LIN {X 0,Y 55.699,Z 480.431,A -85,B 0,C 180,E1 -29739.752,E2 -29739.752} C_VEL
LIN {X 0,Y 58.966,Z 465.331,A -85,B 0,C 180,E1 -29745.097,E2 -29745.097} C_VEL
LIN {X 0,Y 62.169,Z 448.108,A -85,B 0,C 180,E1 -29749.414,E2 -29749.414} C_VEL
LIN {X 0,Y 73.218,Z 385.483,A -85,B 0,C 180,E1 -29760.921,E2 -29760.921} C_VEL
LIN {X 0,Y 72.492,Z 382.499,A -85,B 0,C 180,E1 -29761.896,E2 -29761.896} C_VEL
LIN {X 0,Y 69.464,Z 373.63,A -85,B 0,C 180,E1 -29765.325,E2 -29765.325} C_VEL
LIN {X 0,Y 67.284,Z 368.876,A -85,B 0,C 180,E1 -29767.632,E2 -29767.632} C_VEL
LIN {X 0,Y 64.336,Z 364.78,A -85,B 0,C 180,E1 -29770.407,E2 -29770.407} C_VEL
LIN {X 0,Y 57.379,Z 355.76,A -85,B 0,C 180,E1 -29778.129,E2 -29778.129} C_VEL
LIN {X 0,Y 55.471,Z 351.155,A -85,B 0,C 180,E1 -29781.461,E2 -29781.461} C_VEL
LIN {X 0,Y 51.666,Z 340.966,A -85,B 0,C 180,E1 -29789.989,E2 -29789.989} C_VEL
LIN {X 0,Y 48.729,Z 333.984,A -85,B 0,C 180,E1 -29798.281,E2 -29798.281} C_VEL
LIN {X 0,Y 46.247,Z 330.846,A -85,B 0,C 180,E1 -29805.867,E2 -29805.867} C_VEL
LIN {X 0,Y 45.665,Z 329.617,A -85,B 0,C 180,E1 -29808.495,E2 -29808.495} C_VEL
LIN {X 0,Y 42.859,Z 326.9,A -85,B 0,C 180,E1 -29824.939,E2 -29824.939} C_VEL
LIN {X 0,Y 42.565,Z 326.431,A -85,B 0,C 180,E1 -29831.316,E2 -29831.316} C_VEL
LIN {X 0,Y 42.67,Z 326.804,A -85,B 0,C 180,E1 -29840.533,E2 -29840.533} C_VEL
LIN {X 0,Y 43.226,Z 327.728,A -85,B 0,C 180,E1 -29847.197,E2 -29847.197} C_VEL
LIN {X 0,Y 45.942,Z 330.085,A -85,B 0,C 180,E1 -29860.528,E2 -29860.528} C_VEL
LIN {X 0,Y 47.787,Z 333.251,A -85,B 0,C 180,E1 -29867.187,E2 -29867.187} C_VEL
LIN {X 0,Y 49.086,Z 334.684,A -85,B 0,C 180,E1 -29870.587,E2 -29870.587} C_VEL
LIN {X 0,Y 51.573,Z 340.348,A -85,B 0,C 180,E1 -29877.378,E2 -29877.378} C_VEL
LIN {X 0,Y 55.316,Z 350.367,A -85,B 0,C 180,E1 -29885.909,E2 -29885.909} C_VEL
LIN {X 0,Y 59.591,Z 363.131,A -85,B 0,C 180,E1 -29893.866,E2 -29893.866} C_VEL
LIN {X 0,Y 63.329,Z 378.635,A -85,B 0,C 180,E1 -29900.74,E2 -29900.74} C_VEL
LIN {X 0,Y 67.376,Z 395.193,A -85,B 0,C 180,E1 -29906.947,E2 -29906.947} C_VEL
LIN {X 0,Y 54.893,Z 463.552,A -85,B 0,C 180,E1 -29921.285,E2 -29921.285} C_VEL
LIN {X 0,Y 51.895,Z 478.587,A -85,B 0,C 180,E1 -29926.34,E2 -29926.34} C_VEL
LIN {X 0,Y 48.679,Z 493.737,A -85,B 0,C 180,E1 -29933.463,E2 -29933.463} C_VEL
LIN {X 0,Y 45.63,Z 509.372,A -85,B 0,C 180,E1 -29943.73,E2 -29943.73} C_VEL
LIN {X 0,Y 44.068,Z 522.69,A -85,B 0,C 180,E1 -29955.453,E2 -29955.453} C_VEL
LIN {X 0,Y 44.336,Z 534.77,A -85,B 0,C 180,E1 -29968.467,E2 -29968.467} C_VEL
LIN {X 0,Y 46.533,Z 544.973,A -85,B 0,C 180,E1 -29980.894,E2 -29980.894} C_VEL
LIN {X 0,Y 48.842,Z 550.837,A -85,B 0,C 180,E1 -29988.592,E2 -29988.592} C_VEL
LIN {X 0,Y 49.64,Z 553.845,A -85,B 0,C 180,E1 -29995.146,E2 -29995.146} C_VEL
LIN {X 0,Y 53.747,Z 560.113,A -85,B 0,C 180,E1 -30010.842,E2 -30010.842} C_VEL
LIN {X 0,Y 54.729,Z 560.872,A -85,B 0,C 180,E1 -30015.059,E2 -30015.059} C_VEL
LIN {X 0,Y 46.975,Z 550.464,A -85,B 0,C 180,E1 -30030.899,E2 -30030.899} C_VEL
LIN {X 0,Y 44.588,Z 544.97,A -85,B 0,C 180,E1 -30039.221,E2 -30039.221} C_VEL
LIN {X 0,Y 42.294,Z 536.859,A -85,B 0,C 180,E1 -30050.427,E2 -30050.427} C_VEL
LIN {X 0,Y 41.213,Z 525.272,A -85,B 0,C 180,E1 -30064.884,E2 -30064.884} C_VEL
LIN {X 0,Y 42.221,Z 511.198,A -85,B 0,C 180,E1 -30079.438,E2 -30079.438} C_VEL
LIN {X 0,Y 45.13,Z 495.507,A -85,B 0,C 180,E1 -30091.699,E2 -30091.699} C_VEL
LIN {X 0,Y 48.94,Z 478.571,A -85,B 0,C 180,E1 -30101.013,E2 -30101.013} C_VEL
LIN {X 0,Y 52.42,Z 462.754,A -85,B 0,C 180,E1 -30107.03,E2 -30107.03} C_VEL
LIN {X 0,Y 56.128,Z 443.14,A -85,B 0,C 180,E1 -30112.214,E2 -30112.214} C_VEL
LIN {X 0,Y 66.667,Z 386.304,A -85,B 0,C 180,E1 -30123.427,E2 -30123.427} C_VEL
LIN {X 0,Y 60.039,Z 364.937,A -85,B 0,C 180,E1 -30133.113,E2 -30133.113} C_VEL
LIN {X 0,Y 56.099,Z 352.921,A -85,B 0,C 180,E1 -30140.227,E2 -30140.227} C_VEL
LIN {X 0,Y 55.471,Z 351.155,A -85,B 0,C 180,E1 -30141.461,E2 -30141.461} C_VEL
LIN {X 0,Y 54.149,Z 348.336,A -85,B 0,C 180,E1 -30143.904,E2 -30143.904} C_VEL
LIN {X 0,Y 52.232,Z 346.304,A -85,B 0,C 180,E1 -30146.934,E2 -30146.934} C_VEL
LIN {X 0,Y 46.327,Z 341.623,A -85,B 0,C 180,E1 -30158.375,E2 -30158.375} C_VEL
LIN {X 0,Y 45.874,Z 340.912,A -85,B 0,C 180,E1 -30159.735,E2 -30159.735} C_VEL
LIN {X 0,Y 45.049,Z 339.451,A -85,B 0,C 180,E1 -30162.557,E2 -30162.557} C_VEL
LIN {X 0,Y 43.071,Z 336.15,A -85,B 0,C 180,E1 -30170.881,E2 -30170.881} C_VEL
LIN {X 0,Y 40.853,Z 333.573,A -85,B 0,C 180,E1 -30187.874,E2 -30187.874} C_VEL
LIN {X 0,Y 40.719,Z 333.35,A -85,B 0,C 180,E1 -30193.642,E2 -30193.642} C_VEL
LIN {X 0,Y 41.056,Z 333.988,A -85,B 0,C 180,E1 -30203.361,E2 -30203.361} C_VEL
LIN {X 0,Y 43.333,Z 336.653,A -85,B 0,C 180,E1 -30218.203,E2 -30218.203} C_VEL
LIN {X 0,Y 45.356,Z 339.979,A -85,B 0,C 180,E1 -30226.322,E2 -30226.322} C_VEL
LIN {X 0,Y 46.092,Z 341.294,A -85,B 0,C 180,E1 -30228.723,E2 -30228.723} C_VEL
LIN {X 0,Y 48.368,Z 347.727,A -85,B 0,C 180,E1 -30236.318,E2 -30236.318} C_VEL
LIN {X 0,Y 51.301,Z 357.024,A -85,B 0,C 180,E1 -30244.306,E2 -30244.306} C_VEL
LIN {X 0,Y 54.68,Z 368.265,A -85,B 0,C 180,E1 -30251.748,E2 -30251.748} C_VEL
LIN {X 0,Y 59.813,Z 392.087,A -85,B 0,C 180,E1 -30262.664,E2 -30262.664} C_VEL
LIN {X 0,Y 60.736,Z 395.951,A -85,B 0,C 180,E1 -30264.231,E2 -30264.231} C_VEL
LIN {X 0,Y 48.122,Z 462.205,A -85,B 0,C 180,E1 -30279.548,E2 -30279.548} C_VEL
LIN {X 0,Y 44.955,Z 477.483,A -85,B 0,C 180,E1 -30285.309,E2 -30285.309} C_VEL
LIN {X 0,Y 41.591,Z 492.983,A -85,B 0,C 180,E1 -30293.759,E2 -30293.759} C_VEL
LIN {X 0,Y 38.707,Z 508.521,A -85,B 0,C 180,E1 -30305.932,E2 -30305.932} C_VEL
LIN {X 0,Y 37.602,Z 521.263,A -85,B 0,C 180,E1 -30319.243,E2 -30319.243} C_VEL
LIN {X 0,Y 38.441,Z 532.103,A -85,B 0,C 180,E1 -30332.634,E2 -30332.634} C_VEL
LIN {X 0,Y 41.041,Z 541.3,A -85,B 0,C 180,E1 -30344.898,E2 -30344.898} C_VEL
LIN {X 0,Y 43.949,Z 547.593,A -85,B 0,C 180,E1 -30353.578,E2 -30353.578} C_VEL
LIN {X 0,Y 45.292,Z 550.922,A -85,B 0,C 180,E1 -30361.936,E2 -30361.936} C_VEL
LIN {X 0,Y 46.545,Z 552.86,A -85,B 0,C 180,E1 -30367.17,E2 -30367.17} C_VEL
LIN {X 0,Y 48.338,Z 554.843,A -85,B 0,C 180,E1 -30373.359,E2 -30373.359} C_VEL
LIN {X 0,Y 41.402,Z 545.488,A -85,B 0,C 180,E1 -30388.1,E2 -30388.1} C_VEL
LIN {X 0,Y 38.272,Z 538.77,A -85,B 0,C 180,E1 -30398.444,E2 -30398.444} C_VEL
LIN {X 0,Y 35.716,Z 529.842,A -85,B 0,C 180,E1 -30411.507,E2 -30411.507} C_VEL
LIN {X 0,Y 34.889,Z 518.192,A -85,B 0,C 180,E1 -30427.223,E2 -30427.223} C_VEL
LIN {X 0,Y 36.013,Z 505.529,A -85,B 0,C 180,E1 -30441.454,E2 -30441.454} C_VEL
LIN {X 0,Y 38.612,Z 492.029,A -85,B 0,C 180,E1 -30453.086,E2 -30453.086} C_VEL
LIN {X 0,Y 42.449,Z 475.565,A -85,B 0,C 180,E1 -30463.064,E2 -30463.064} C_VEL
LIN {X 0,Y 46.079,Z 459.423,A -85,B 0,C 180,E1 -30469.683,E2 -30469.683} C_VEL
LIN {X 0,Y 51.287,Z 432.312,A -85,B 0,C 180,E1 -30477.057,E2 -30477.057} C_VEL
LIN {X 0,Y 60.147,Z 387.558,A -85,B 0,C 180,E1 -30486.307,E2 -30486.307} C_VEL
LIN {X 0,Y 54.234,Z 367.063,A -85,B 0,C 180,E1 -30496.882,E2 -30496.882} C_VEL
LIN {X 0,Y 50.513,Z 354.677,A -85,B 0,C 180,E1 -30505.432,E2 -30505.432} C_VEL
LIN {X 0,Y 47.276,Z 344.825,A -85,B 0,C 180,E1 -30514.818,E2 -30514.818} C_VEL
LIN {X 0,Y 45.874,Z 340.912,A -85,B 0,C 180,E1 -30519.735,E2 -30519.735} C_VEL
LIN {X 0,Y 44.694,Z 339.743,A -85,B 0,C 180,E1 -30523.229,E2 -30523.229} C_VEL
LIN {X 0,Y 42.755,Z 339.599,A -85,B 0,C 180,E1 -30528.729,E2 -30528.729} C_VEL
LIN {X 0,Y 39.587,Z 340.945,A -85,B 0,C 180,E1 -30541.368,E2 -30541.368} C_VEL
LIN {X 0,Y 39.05,Z 340.575,A -85,B 0,C 180,E1 -30547.31,E2 -30547.31} C_VEL
LIN {X 0,Y 38.927,Z 340.263,A -85,B 0,C 180,E1 -30556.212,E2 -30556.212} C_VEL
LIN {X 0,Y 39.266,Z 341.215,A -85,B 0,C 180,E1 -30564.444,E2 -30564.444} C_VEL
LIN {X 0,Y 40.791,Z 343.118,A -85,B 0,C 180,E1 -30575.645,E2 -30575.645} C_VEL
LIN {X 0,Y 42.632,Z 346.581,A -85,B 0,C 180,E1 -30584.499,E2 -30584.499} C_VEL
LIN {X 0,Y 44.258,Z 352.215,A -85,B 0,C 180,E1 -30591.784,E2 -30591.784} C_VEL
LIN {X 0,Y 46.576,Z 361.026,A -85,B 0,C 180,E1 -30600.249,E2 -30600.249} C_VEL
LIN {X 0,Y 49.278,Z 371.489,A -85,B 0,C 180,E1 -30608.031,E2 -30608.031} C_VEL
LIN {X 0,Y 54.241,Z 396.884,A -85,B 0,C 180,E1 -30621.036,E2 -30621.036} C_VEL
LIN {X 0,Y 41.251,Z 461.358,A -85,B 0,C 180,E1 -30637.528,E2 -30637.528} C_VEL
LIN {X 0,Y 37.971,Z 476.59,A -85,B 0,C 180,E1 -30644.196,E2 -30644.196} C_VEL
LIN {X 0,Y 34.373,Z 492.897,A -85,B 0,C 180,E1 -30654.885,E2 -30654.885} C_VEL
LIN {X 0,Y 31.868,Z 507.771,A -85,B 0,C 180,E1 -30669.389,E2 -30669.389} C_VEL
LIN {X 0,Y 31.573,Z 521.341,A -85,B 0,C 180,E1 -30686.827,E2 -30686.827} C_VEL
LIN {X 0,Y 34.309,Z 533.798,A -85,B 0,C 180,E1 -30704.852,E2 -30704.852} C_VEL
LIN {X 0,Y 38.424,Z 542.459,A -85,B 0,C 180,E1 -30717.226,E2 -30717.226} C_VEL
LIN {X 0,Y 39.378,Z 544.025,A -85,B 0,C 180,E1 -30719.409,E2 -30719.409} C_VEL
LIN {X 0,Y 41.749,Z 547.874,A -85,B 0,C 180,E1 -30730.064,E2 -30730.064} C_VEL
LIN {X 0,Y 40.899,Z 546.914,A -85,B 0,C 180,E1 -30733.439,E2 -30733.439} C_VEL
LIN {X 0,Y 36.103,Z 540.296,A -85,B 0,C 180,E1 -30744.258,E2 -30744.258} C_VEL
LIN {X 0,Y 31.953,Z 531.995,A -85,B 0,C 180,E1 -30757.352,E2 -30757.352} C_VEL
LIN {X 0,Y 29.008,Z 520.124,A -85,B 0,C 180,E1 -30776.173,E2 -30776.173} C_VEL
LIN {X 0,Y 28.986,Z 506.448,A -85,B 0,C 180,E1 -30795.818,E2 -30795.818} C_VEL
LIN {X 0,Y 31.436,Z 491.666,A -85,B 0,C 180,E1 -30812.059,E2 -30812.059} C_VEL
LIN {X 0,Y 35.319,Z 475.268,A -85,B 0,C 180,E1 -30824.13,E2 -30824.13} C_VEL
LIN {X 0,Y 39.112,Z 459.245,A -85,B 0,C 180,E1 -30831.813,E2 -30831.813} C_VEL
LIN {X 0,Y 44.134,Z 434.472,A -85,B 0,C 180,E1 -30839.454,E2 -30839.454} C_VEL
LIN {X 0,Y 53.774,Z 388.856,A -85,B 0,C 180,E1 -30849.754,E2 -30849.754} C_VEL
LIN {X 0,Y 48.635,Z 369.267,A -85,B 0,C 180,E1 -30861.418,E2 -30861.418} C_VEL
LIN {X 0,Y 45.694,Z 357.878,A -85,B 0,C 180,E1 -30870.431,E2 -30870.431} C_VEL
LIN {X 0,Y 43.259,Z 349.06,A -85,B 0,C 180,E1 -30880.051,E2 -30880.051} C_VEL
LIN {X 0,Y 42.294,Z 345.754,A -85,B 0,C 180,E1 -30884.915,E2 -30884.915} C_VEL
LIN {X 0,Y 40.496,Z 342.589,A -85,B 0,C 180,E1 -30893.963,E2 -30893.963} C_VEL
LIN {X 0,Y 39.05,Z 340.575,A -85,B 0,C 180,E1 -30907.31,E2 -30907.31} C_VEL
LIN {X 0,Y 38.873,Z 340.516,A -85,B 0,C 180,E1 -30911.953,E2 -30911.953} C_VEL
LIN {X 0,Y 38.514,Z 342.149,A -85,B 0,C 180,E1 -30918.235,E2 -30918.235} C_VEL
LIN {X 0,Y 38.656,Z 350.53,A -85,B 0,C 180,E1 -30935.353,E2 -30935.353} C_VEL
LIN {X 0,Y 39.495,Z 352.402,A -85,B 0,C 180,E1 -30940.278,E2 -30940.278} C_VEL
LIN {X 0,Y 40.487,Z 357.291,A -85,B 0,C 180,E1 -30947.128,E2 -30947.128} C_VEL
LIN {X 0,Y 42.133,Z 365.385,A -85,B 0,C 180,E1 -30955.682,E2 -30955.682} C_VEL
LIN {X 0,Y 44.089,Z 374.602,A -85,B 0,C 180,E1 -30963.471,E2 -30963.471} C_VEL
LIN {X 0,Y 47.888,Z 397.772,A -85,B 0,C 180,E1 -30977.075,E2 -30977.075} C_VEL
LIN {X 0,Y 34.48,Z 460.293,A -85,B 0,C 180,E1 -30994.776,E2 -30994.776} C_VEL
LIN {X 0,Y 30.855,Z 476.275,A -85,B 0,C 180,E1 -31003.118,E2 -31003.118} C_VEL
LIN {X 0,Y 27.378,Z 491.75,A -85,B 0,C 180,E1 -31015.801,E2 -31015.801} C_VEL
LIN {X 0,Y 25.279,Z 506.325,A -85,B 0,C 180,E1 -31033.881,E2 -31033.881} C_VEL
LIN {X 0,Y 26.119,Z 520.123,A -85,B 0,C 180,E1 -31055.812,E2 -31055.812} C_VEL
LIN {X 0,Y 30.055,Z 531.553,A -85,B 0,C 180,E1 -31074.175,E2 -31074.175} C_VEL
LIN {X 0,Y 35.361,Z 540.233,A -85,B 0,C 180,E1 -31086.621,E2 -31086.621} C_VEL
LIN {X 0,Y 35.762,Z 540.823,A -85,B 0,C 180,E1 -31088.165,E2 -31088.165} C_VEL
LIN {X 0,Y 34.756,Z 539.691,A -85,B 0,C 180,E1 -31091.272,E2 -31091.272} C_VEL
LIN {X 0,Y 29.811,Z 532.795,A -85,B 0,C 180,E1 -31101.937,E2 -31101.937} C_VEL
LIN {X 0,Y 24.888,Z 522.545,A -85,B 0,C 180,E1 -31118.961,E2 -31118.961} C_VEL
LIN {X 0,Y 22.631,Z 512.196,A -85,B 0,C 180,E1 -31137.761,E2 -31137.761} C_VEL
LIN {X 0,Y 23.065,Z 498.236,A -85,B 0,C 180,E1 -31160.979,E2 -31160.979} C_VEL
LIN {X 0,Y 25.842,Z 484.236,A -85,B 0,C 180,E1 -31177.712,E2 -31177.712} C_VEL
LIN {X 0,Y 29.891,Z 468.405,A -85,B 0,C 180,E1 -31189.814,E2 -31189.814} C_VEL
LIN {X 0,Y 34.008,Z 451.104,A -85,B 0,C 180,E1 -31197.761,E2 -31197.761} C_VEL
LIN {X 0,Y 43.278,Z 408.433,A -85,B 0,C 180,E1 -31210.219,E2 -31210.219} C_VEL
LIN {X 0,Y 47.526,Z 389.835,A -85,B 0,C 180,E1 -31214.114,E2 -31214.114} C_VEL
LIN {X 0,Y 43.475,Z 372.281,A -85,B 0,C 180,E1 -31226.327,E2 -31226.327} C_VEL
LIN {X 0,Y 41.397,Z 362.028,A -85,B 0,C 180,E1 -31235.507,E2 -31235.507} C_VEL
LIN {X 0,Y 39.726,Z 353.828,A -85,B 0,C 180,E1 -31245.506,E2 -31245.506} C_VEL
LIN {X 0,Y 39.104,Z 351.342,A -85,B 0,C 180,E1 -31249.831,E2 -31249.831} C_VEL
LIN {X 0,Y 38.157,Z 349.166,A -85,B 0,C 180,E1 -31256.639,E2 -31256.639} C_VEL
LIN {X 0,Y 37.16,Z 347.153,A -85,B 0,C 180,E1 -31270.856,E2 -31270.856} C_VEL
LIN {X 0,Y 37.194,Z 347.447,A -85,B 0,C 180,E1 -31279.787,E2 -31279.787} C_VEL
LIN {X 0,Y 38.336,Z 349.624,A -85,B 0,C 180,E1 -31292.811,E2 -31292.811} C_VEL
LIN {X 0,Y 38.656,Z 350.53,A -85,B 0,C 180,E1 -31295.353,E2 -31295.353} C_VEL
LIN {X 0,Y 38.999,Z 352.639,A -85,B 0,C 180,E1 -31298.856,E2 -31298.856} C_VEL
LIN {X 0,Y 38.868,Z 356.651,A -85,B 0,C 180,E1 -31302.151,E2 -31302.151} C_VEL
LIN {X 0,Y 37.771,Z 367.083,A -85,B 0,C 180,E1 -31307.767,E2 -31307.767} C_VEL
LIN {X 0,Y 37.935,Z 369.465,A -85,B 0,C 180,E1 -31309.947,E2 -31309.947} C_VEL
LIN {X 0,Y 39.215,Z 378.078,A -85,B 0,C 180,E1 -31318.1,E2 -31318.1} C_VEL
LIN {X 0,Y 41.811,Z 398.741,A -85,B 0,C 180,E1 -31332.14,E2 -31332.14} C_VEL
LIN {X 0,Y 27.566,Z 460.093,A -85,B 0,C 180,E1 -31351.321,E2 -31351.321} C_VEL
LIN {X 0,Y 24.111,Z 474.417,A -85,B 0,C 180,E1 -31360.392,E2 -31360.392} C_VEL
LIN {X 0,Y 20.594,Z 489.602,A -85,B 0,C 180,E1 -31376.353,E2 -31376.353} C_VEL
LIN {X 0,Y 19.004,Z 505.025,A -85,B 0,C 180,E1 -31402.058,E2 -31402.058} C_VEL
LIN {X 0,Y 21.266,Z 517.608,A -85,B 0,C 180,E1 -31426.835,E2 -31426.835} C_VEL
LIN {X 0,Y 27.013,Z 529.325,A -85,B 0,C 180,E1 -31446.311,E2 -31446.311} C_VEL
LIN {X 0,Y 27.413,Z 530.079,A -85,B 0,C 180,E1 -31449.709,E2 -31449.709} C_VEL
LIN {X 0,Y 20.751,Z 519.361,A -85,B 0,C 180,E1 -31466.59,E2 -31466.59} C_VEL
LIN {X 0,Y 16.822,Z 507.591,A -85,B 0,C 180,E1 -31490.967,E2 -31490.967} C_VEL
LIN {X 0,Y 16.744,Z 493.859,A -85,B 0,C 180,E1 -31520.823,E2 -31520.823} C_VEL
LIN {X 0,Y 20.143,Z 477.936,A -85,B 0,C 180,E1 -31544.229,E2 -31544.229} C_VEL
LIN {X 0,Y 24.2,Z 463.204,A -85,B 0,C 180,E1 -31556.209,E2 -31556.209} C_VEL
LIN {X 0,Y 29.016,Z 443.606,A -85,B 0,C 180,E1 -31565.244,E2 -31565.244} C_VEL
LIN {X 0,Y 41.614,Z 391.315,A -85,B 0,C 180,E1 -31579.319,E2 -31579.319} C_VEL
LIN {X 0,Y 38.701,Z 375.439,A -85,B 0,C 180,E1 -31592.22,E2 -31592.22} C_VEL
LIN {X 0,Y 37.391,Z 365.643,A -85,B 0,C 180,E1 -31602.258,E2 -31602.258} C_VEL
LIN {X 0,Y 36.522,Z 358.107,A -85,B 0,C 180,E1 -31612.619,E2 -31612.619} C_VEL
LIN {X 0,Y 36.212,Z 356.647,A -85,B 0,C 180,E1 -31616.172,E2 -31616.172} C_VEL
LIN {X 0,Y 35.789,Z 355.49,A -85,B 0,C 180,E1 -31620.66,E2 -31620.66} C_VEL
LIN {X 0,Y 35.342,Z 354.009,A -85,B 0,C 180,E1 -31631.845,E2 -31631.845} C_VEL
LIN {X 0,Y 35.319,Z 354.329,A -85,B 0,C 180,E1 -31638.53,E2 -31638.53} C_VEL
LIN {X 0,Y 36.02,Z 356.088,A -85,B 0,C 180,E1 -31649.755,E2 -31649.755} C_VEL
LIN {X 0,Y 36.582,Z 358.243,A -85,B 0,C 180,E1 -31655.654,E2 -31655.654} C_VEL
LIN {X 0,Y 37.254,Z 364.143,A -85,B 0,C 180,E1 -31663.931,E2 -31663.931} C_VEL
LIN {X 0,Y 37.935,Z 369.465,A -85,B 0,C 180,E1 -31669.947,E2 -31669.947} C_VEL
LIN {X 0,Y 38.25,Z 372.81,A -85,B 0,C 180,E1 -31672.956,E2 -31672.956} C_VEL
LIN {X 0,Y 38.048,Z 378.32,A -85,B 0,C 180,E1 -31676.137,E2 -31676.137} C_VEL
LIN {X 0,Y 35.891,Z 395.74,A -85,B 0,C 180,E1 -31683.196,E2 -31683.196} C_VEL
LIN {X 0,Y 36.007,Z 399.484,A -85,B 0,C 180,E1 -31685.572,E2 -31685.572} C_VEL
LIN {X 0,Y 21.782,Z 456.042,A -85,B 0,C 180,E1 -31703.784,E2 -31703.784} C_VEL
LIN {X 0,Y 17.915,Z 470.789,A -85,B 0,C 180,E1 -31714.119,E2 -31714.119} C_VEL
LIN {X 0,Y 14.013,Z 486.395,A -85,B 0,C 180,E1 -31735.699,E2 -31735.699} C_VEL
LIN {X 0,Y 13.341,Z 502.281,A -85,B 0,C 180,E1 -31774.195,E2 -31774.195} C_VEL
LIN {X 0,Y 17.376,Z 514.384,A -85,B 0,C 180,E1 -31802.24,E2 -31802.24} C_VEL
LIN {X 0,Y 18.166,Z 516.143,A -85,B 0,C 180,E1 -31809.28,E2 -31809.28} C_VEL
LIN {X 0,Y 12.488,Z 505.357,A -85,B 0,C 180,E1 -31830.47,E2 -31830.47} C_VEL
LIN {X 0,Y 10.277,Z 491.044,A -85,B 0,C 180,E1 -31874.828,E2 -31874.828} C_VEL
LIN {X 0,Y 13.466,Z 475.925,A -85,B 0,C 180,E1 -31908.979,E2 -31908.979} C_VEL
LIN {X 0,Y 18.259,Z 460.035,A -85,B 0,C 180,E1 -31924.659,E2 -31924.659} C_VEL
LIN {X 0,Y 23.728,Z 439.65,A -85,B 0,C 180,E1 -31934.233,E2 -31934.233} C_VEL
LIN {X 0,Y 36.018,Z 392.57,A -85,B 0,C 180,E1 -31946.31,E2 -31946.31} C_VEL
LIN {X 0,Y 34.379,Z 378.369,A -85,B 0,C 180,E1 -31959.796,E2 -31959.796} C_VEL
LIN {X 0,Y 33.915,Z 369.45,A -85,B 0,C 180,E1 -31970.18,E2 -31970.18} C_VEL
LIN {X 0,Y 33.891,Z 362.955,A -85,B 0,C 180,E1 -31979.907,E2 -31979.907} C_VEL
LIN {X 0,Y 33.648,Z 361.974,A -85,B 0,C 180,E1 -31984.321,E2 -31984.321} C_VEL
LIN {X 0,Y 33.513,Z 360.869,A -85,B 0,C 180,E1 -31994.709,E2 -31994.709} C_VEL
LIN {X 0,Y 33.81,Z 362.645,A -85,B 0,C 180,E1 -32006.52,E2 -32006.52} C_VEL
LIN {X 0,Y 33.932,Z 364.078,A -85,B 0,C 180,E1 -32010.209,E2 -32010.209} C_VEL
LIN {X 0,Y 34.085,Z 372.286,A -85,B 0,C 180,E1 -32021.421,E2 -32021.421} C_VEL
LIN {X 0,Y 34.672,Z 381.101,A -85,B 0,C 180,E1 -32031.025,E2 -32031.025} C_VEL
LIN {X 0,Y 36.007,Z 399.484,A -85,B 0,C 180,E1 -32045.572,E2 -32045.572} C_VEL
LIN {X 0,Y 35.797,Z 403.072,A -85,B 0,C 180,E1 -32047.31,E2 -32047.31} C_VEL
LIN {X 0,Y 34.709,Z 406.705,A -85,B 0,C 180,E1 -32047.875,E2 -32047.875} C_VEL
LIN {X 0,Y 33.026,Z 410.274,A -85,B 0,C 180,E1 -32047.575,E2 -32047.575} C_VEL
LIN {X 0,Y 25.461,Z 422.468,A -85,B 0,C 180,E1 -32043.062,E2 -32043.062} C_VEL
LIN {X 0,Y 23.309,Z 427.207,A -85,B 0,C 180,E1 -32042.389,E2 -32042.389} C_VEL
LIN {X 0,Y 22.982,Z 428.195,A -85,B 0,C 180,E1 -32042.523,E2 -32042.523} C_VEL
LIN {X 0,Y 14.366,Z 459.493,A -85,B 0,C 180,E1 -32055.75,E2 -32055.75} C_VEL
LIN {X 0,Y 9.832,Z 474.185,A -85,B 0,C 180,E1 -32072.024,E2 -32072.024} C_VEL
LIN {X 0,Y 6.827,Z 488.219,A -85,B 0,C 180,E1 -32115.17,E2 -32115.17} C_VEL
LIN {X 0,Y 8.615,Z 498.324,A -85,B 0,C 180,E1 -32157.107,E2 -32157.107} C_VEL
LIN {X 0,Y 8.634,Z 498.873,A -85,B 0,C 180,E1 -32165.453,E2 -32165.453} C_VEL
LIN {X 0,Y 4.169,Z 484.974,A -85,B 0,C 180,E1 -32232.088,E2 -32232.088} C_VEL
LIN {X 0,Y 8.826,Z 468.856,A -85,B 0,C 180,E1 -32290.042,E2 -32290.042} C_VEL
LIN {X 0,Y 14.668,Z 451.486,A -85,B 0,C 180,E1 -32302.234,E2 -32302.234} C_VEL
LIN {X 0,Y 25.965,Z 411.813,A -85,B 0,C 180,E1 -32312.989,E2 -32312.989} C_VEL
LIN {X 0,Y 31.081,Z 393.528,A -85,B 0,C 180,E1 -32315.7,E2 -32315.7} C_VEL
LIN {X 0,Y 30.804,Z 379.395,A -85,B 0,C 180,E1 -32331.418,E2 -32331.418} C_VEL
LIN {X 0,Y 31.316,Z 371.449,A -85,B 0,C 180,E1 -32342.33,E2 -32342.33} C_VEL
LIN {X 0,Y 31.698,Z 368.71,A -85,B 0,C 180,E1 -32346.558,E2 -32346.558} C_VEL
LIN {X 0,Y 31.66,Z 367.961,A -85,B 0,C 180,E1 -32355.184,E2 -32355.184} C_VEL
LIN {X 0,Y 31.668,Z 369.074,A -85,B 0,C 180,E1 -32362.262,E2 -32362.262} C_VEL
LIN {X 0,Y 30.946,Z 376.582,A -85,B 0,C 180,E1 -32372.997,E2 -32372.997} C_VEL
LIN {X 0,Y 30.741,Z 384.045,A -85,B 0,C 180,E1 -32381.976,E2 -32381.976} C_VEL
LIN {X 0,Y 30.786,Z 400.426,A -85,B 0,C 180,E1 -32397.008,E2 -32397.008} C_VEL
LIN {X 0,Y 22.982,Z 428.195,A -85,B 0,C 180,E1 -32402.523,E2 -32402.523} C_VEL
LIN {X 0,Y 20.868,Z 433.722,A -85,B 0,C 180,E1 -32402.627,E2 -32402.627} C_VEL
LIN {X 0,Y 11.95,Z 451.239,A -85,B 0,C 180,E1 -32393.149,E2 -32393.149} C_VEL
LIN {X 0,Y 9.771,Z 456.734,A -85,B 0,C 180,E1 -32391.698,E2 -32391.698} C_VEL
LIN {X 0,Y 4.248,Z 471.603,A -85,B 0,C 180,E1 -32398.807,E2 -32398.807} C_VEL
LIN {X 0,Y 2.908,Z 474.679,A -85,B 0,C 180,E1 -32402.943,E2 -32402.943} C_VEL
LIN {X 0,Y 1.85,Z 476.41,A -85,B 0,C 180,E1 -32400.17,E2 -32400.17} C_VEL
LIN {X 0,Y 6.717,Z 461.718,A -85,B 0,C 180,E1 -32333.83,E2 -32333.83} C_VEL
LIN {X 0,Y 12.892,Z 442.722,A -85,B 0,C 180,E1 -32327.528,E2 -32327.528} C_VEL
LIN {X 0,Y 27.135,Z 394.725,A -85,B 0,C 180,E1 -32327.789,E2 -32327.789} C_VEL
LIN {X 0,Y 28.324,Z 382.12,A -85,B 0,C 180,E1 -32343.348,E2 -32343.348} C_VEL
LIN {X 0,Y 29.766,Z 375.089,A -85,B 0,C 180,E1 -32353.464,E2 -32353.464} C_VEL
LIN {X 0,Y 29.664,Z 375.476,A -85,B 0,C 180,E1 -32355.27,E2 -32355.27} C_VEL
LIN {X 0,Y 28.068,Z 384.218,A -85,B 0,C 180,E1 -32367.53,E2 -32367.53} C_VEL
LIN {X 0,Y 26.948,Z 393.457,A -85,B 0,C 180,E1 -32377.385,E2 -32377.385} C_VEL
LIN {X 0,Y 26.346,Z 401.615,A -85,B 0,C 180,E1 -32385.459,E2 -32385.459} C_VEL
LIN {X 0,Y 9.771,Z 456.734,A -85,B 0,C 180,E1 -32391.698,E2 -32391.698} C_VEL
LIN {X 0,Y 9.473,Z 456.001,A -85,B 0,C 180,E1 -32386.95,E2 -32386.95} C_VEL
LIN {X 0,Y 9.896,Z 451.996,A -85,B 0,C 180,E1 -32377.676,E2 -32377.676} C_VEL
LIN {X 0,Y 13.209,Z 437.71,A -85,B 0,C 180,E1 -32365.46,E2 -32365.46} C_VEL
LIN {X 0,Y 15.489,Z 429.211,A -85,B 0,C 180,E1 -32364.426,E2 -32364.426} C_VEL
LIN {X 0,Y 16.302,Z 426.4,A -85,B 0,C 180,E1 -32365.227,E2 -32365.227} C_VEL
LIN {X 0,Y 23.388,Z 402.26,A -85,B 0,C 180,E1 -32370.114,E2 -32370.114} C_VEL
LIN {X 0,Y 26.337,Z 387.922,A -85,B 0,C 180,E1 -32355.227,E2 -32355.227} C_VEL
LIN {X 0,Y 26.54,Z 387.155,A -85,B 0,C 180,E1 -32353.948,E2 -32353.948} C_VEL
LIN {X 0,Y 24.572,Z 396.145,A -85,B 0,C 180,E1 -32342.717,E2 -32342.717} C_VEL
LIN {X 0,Y 12.25,Z 440.44,A -85,B 0,C 180,E1 -32359.029,E2 -32359.029} C_VEL
LIN {X 0,Y 12.521,Z 439.549,A -85,B 0,C 180,E1 -32360.445,E2 -32360.445} C_VEL
LIN {X 0,Y 16.302,Z 426.4,A -85,B 0,C 180,E1 -32365.227,E2 -32365.227} C_VEL
LIN {X 0,Y 20.006,Z 427.005,A -85,B 0,C 180,E1 -32369.165,E2 -32369.165} C_VEL
LIN {X 0,Y 20.006,Z 600,A -85,B 0,C 180,E1 -32369.165,E2 -32369.165} C_VEL
LIN {X 0,Y 20.006,Z 600,A -85,B 0,C 180,E1 -32369.165,E2 -32369.165}

QRS_NEXT_CUT()

QRS_NEXT()
QRS_HOME()

END
